FUNCTION "fc" : Bool
{ S7_Optimized_Access := 'TRUE' }
VERSION : 0.1
   VAR_INPUT
      a : Bool;
   END_VAR


BEGIN
	#fc := NOT #a;
END_FUNCTION

